FUNCTION F_BoomAnimation 
VAR_INPUT
	fScale : LREAL;
	fBoomAngle : LREAL;
	fBoomLength : LREAL;
END_VAR
VAR_OUTPUT
	fBoomTipX : INT;
	fBoomTipY : INT;
END_VAR
VAR
END_VAR

fBoomTipX := LREAL_TO_INT( fBoomLength * ( COS(fBoomAngle) - SIN(fBoomAngle) ) * fScale );
fBoomTipY := LREAL_TO_INT( fBoomLength * ( SIN(fBoomAngle) + COS(fBoomAngle) ) * fScale );

END_FUNCTION

(* stored: Version 1.1.0.1, ProductVersion 3.1.4024.10
   POU F_BoomAnimation: Id {8658192c-b10e-4d47-8f72-6b5a3927997e}, SpecialFunc None *)
